FUNCTION_BLOCK TempParoAcumulad
VAR_INPUT
	EnableCount:BOOL;
	ParoActivo:BOOL;

	DateAndTimeActual:DATE_AND_TIME;
	P_resetCont:BOOL;
	
END_VAR
VAR_OUTPUT
	t_Acumulado:TIME;
END_VAR
VAR
	FlancoUp_Enable:r_trig;
	FlancoDo_Enable:f_trig;
	t_InicioSuma:TIME;
	t_FinSuma:TIME;
END_VAR

FlancoUp_Enable(CLK:=EnableCount);
FlancoDo_Enable(CLK:=EnableCount);

IF FlancoUp_Enable.Q THEN 
	InicioHoraCont();
END_IF
IF FlancoDo_Enable.Q AND ParoActivo THEN  
	FinHoraCont();
END_IF
IF P_resetCont THEN 
	ResetContador();
	P_resetCont:=FALSE;
END_IF

METHOD FinHoraCont : BOOL
VAR_INPUT
END_VAR
t_FinSuma := DT_TO_TIME(DateAndTimeActual);
t_Acumulado:= t_Acumulado + (t_FinSuma-t_InicioSuma);
END_METHOD

METHOD InicioHoraCont : BOOL
VAR_INPUT
END_VAR
t_InicioSuma := DT_TO_TIME(DateAndTimeActual) ;
END_METHOD

METHOD ResetContador : BOOL
VAR_INPUT
END_VAR
InicioHoraCont();
t_Acumulado:=T#0S;
END_METHOD

END_FUNCTION_BLOCK

(* stored: Version 1.1.0.1, ProductVersion 3.1.4024.12
   POU TempParoAcumulad: Id {f3fc6d10-ed21-45d6-875f-84933478080e}, SpecialFunc None
   Method FinHoraCont: Id {1fb14688-e825-4653-9e12-12a2b9dee7b6}
   Method InicioHoraCont: Id {bd5a6f4d-52ae-4248-a9ef-edf3b851718e}
   Method ResetContador: Id {02296109-42f9-4a41-8dae-91f14d975529} *)
